Fanuc TP program (LS listing): BASE_RDY_COND.LS

/PROG  BASE_RDY_COND	  Cond
/ATTR
OWNER		= MNEDITOR;
COMMENT		= "monitor";
PROG_SIZE	= 162;
CREATE		= DATE 25-07-16  TIME 20:25:52;
MODIFIED	= DATE 25-07-16  TIME 20:32:18;
FILE_NAME	= ;
VERSION		= 0;
LINE_COUNT	= 1;
MEMORY_SIZE	= 538;
PROTECT		= READ_WRITE;
TCD:  STACK_SIZE	= 0,
      TASK_PRIORITY	= 50,
      TIME_SLICE	= 0,
      BUSY_LAMP_OFF	= 0,
      ABORT_REQUEST	= 0,
      PAUSE_REQUEST	= 0;
DEFAULT_GROUP	= *,*,*,*,*;
CONTROL_CODE	= 00000000 00000000;
/MN
   1:  WHEN DI[4:ON :robot base rdy]=OFF,CALL BASE_MOVED ;
/POS
/END
